FUNCTION_BLOCK EL_Scale (* Scale: output values from its holder -> outputs (break before make); one holder at a time; all off on release or when the module aborts; inputs -> state channel when they change *)
  (* Standard: 61499-2 *)
  (* Version 0.1, 2026-09-28, Project contributors, AAU Smart Production Lab *)
  PACKAGE filling;
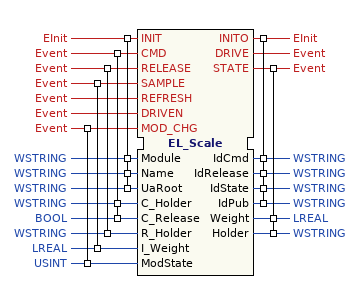
  EVENT_INPUT
    INIT : EInit WITH Module, Name, UaRoot;
    CMD WITH C_Holder, C_Release;
    RELEASE WITH R_Holder;
    SAMPLE WITH I_Weight;
    REFRESH;
    DRIVEN;
    MOD_CHG WITH ModState;
  END_EVENT
  EVENT_OUTPUT
    INITO : EInit WITH IdCmd, IdRelease, IdState, IdPub;
    DRIVE;
    STATE WITH Weight, Holder;
  END_EVENT
  VAR_INPUT
    Module : WSTRING;
    Name : WSTRING;
    UaRoot : WSTRING;
    C_Holder : WSTRING;
    C_Release : BOOL;
    R_Holder : WSTRING;
    I_Weight : LREAL;
    ModState : USINT;
  END_VAR
  VAR_OUTPUT
    IdCmd : WSTRING;
    IdRelease : WSTRING;
    IdState : WSTRING;
    IdPub : WSTRING;
    Weight : LREAL;
    Holder : WSTRING;
  END_VAR
  VAR
    Publish : BOOL;
    Beat : USINT;
    LastHolder : WSTRING;
    Pending : BOOL;
    OffPending : BOOL;
    L_Weight : LREAL;
  END_VAR
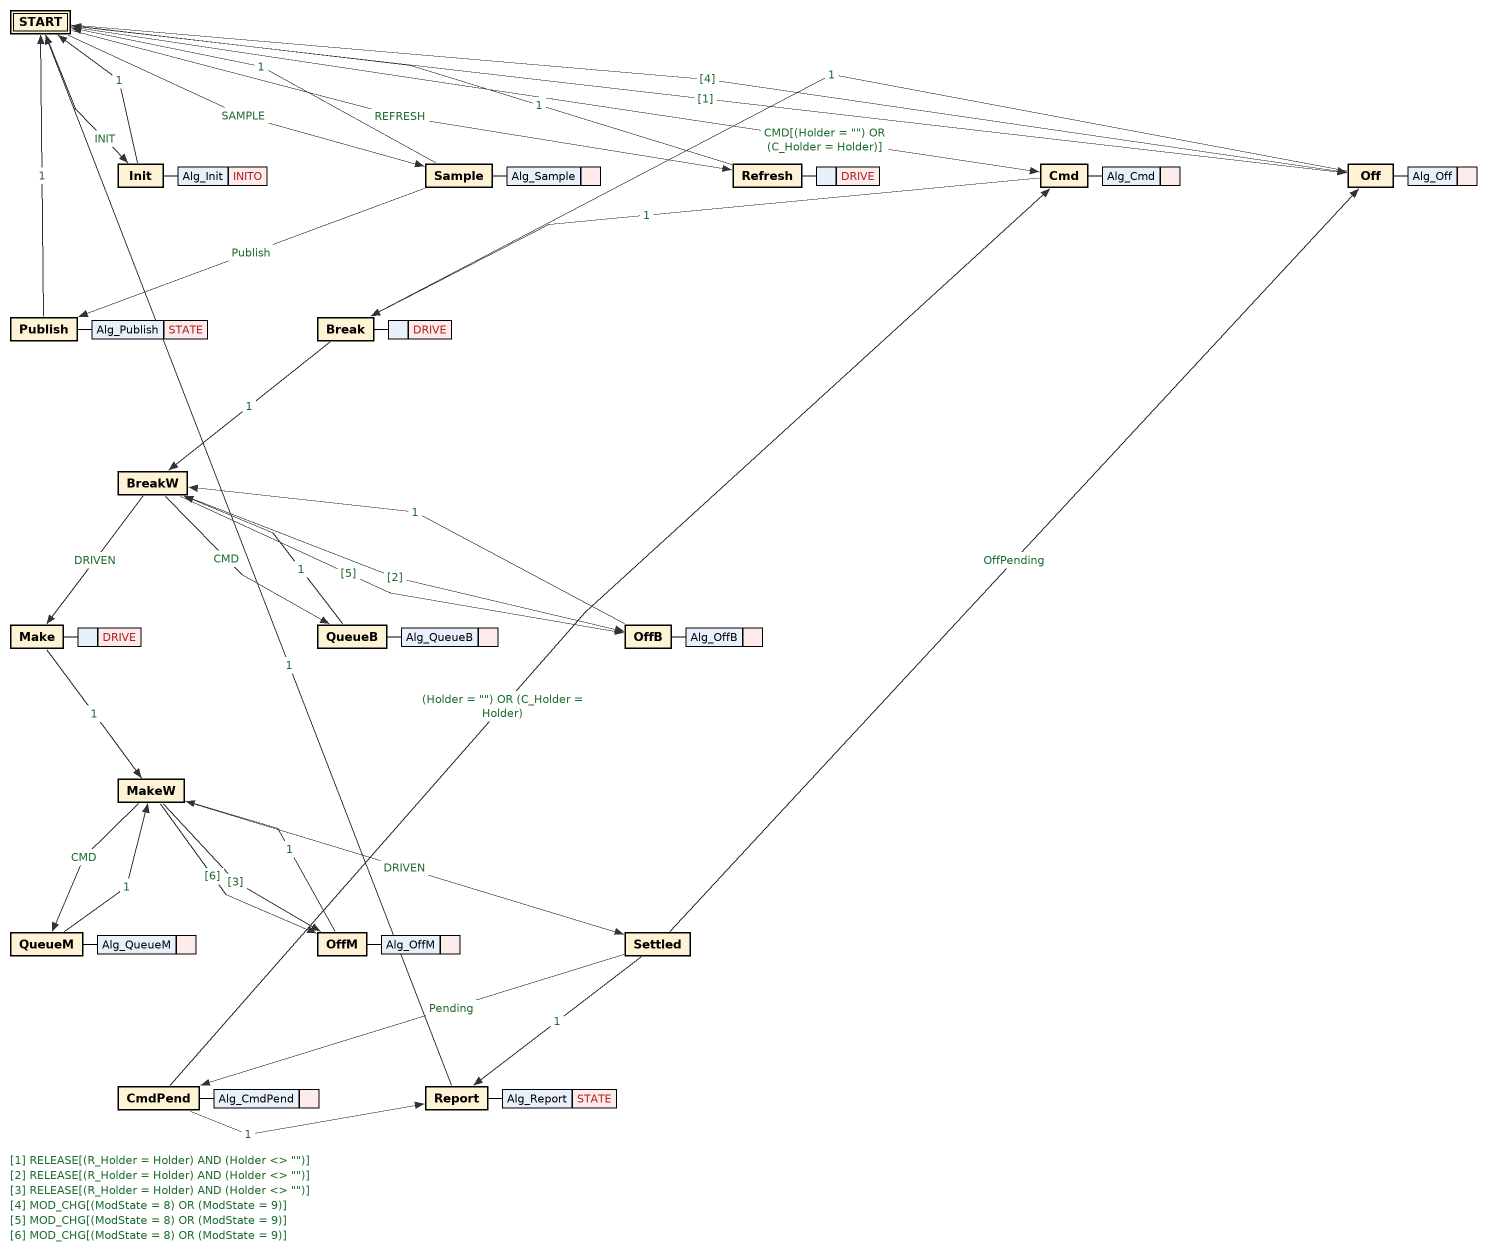
  EC_STATES
    START;
    Init : Alg_Init -> INITO;
    Sample : Alg_Sample;
    Publish : Alg_Publish -> STATE;
    Refresh : -> DRIVE;
    Cmd : Alg_Cmd;
    Off : Alg_Off;
    Break : -> DRIVE;
    Make : -> DRIVE;
    BreakW;
    MakeW;
    QueueB : Alg_QueueB;
    OffB : Alg_OffB;
    QueueM : Alg_QueueM;
    OffM : Alg_OffM;
    CmdPend : Alg_CmdPend;
    Settled;
    Report : Alg_Report -> STATE;
  END_STATES
  EC_TRANSITIONS
    START TO Init := INIT;
    START TO Sample := SAMPLE;
    START TO Refresh := REFRESH;
    START TO Cmd := CMD[(Holder = "") OR (C_Holder = Holder)];
    START TO Off := RELEASE[(R_Holder = Holder) AND (Holder <> "")];
    START TO Off := MOD_CHG[(ModState = 8) OR (ModState = 9)];
    Init TO START := 1;
    Sample TO Publish := Publish;
    Sample TO START := 1;
    Publish TO START := 1;
    Refresh TO START := 1;
    Cmd TO Break := 1;
    Off TO Break := 1;
    Break TO BreakW := 1;
    BreakW TO Make := DRIVEN;
    Make TO MakeW := 1;
    MakeW TO Settled := DRIVEN;
    BreakW TO QueueB := CMD;
    BreakW TO OffB := RELEASE[(R_Holder = Holder) AND (Holder <> "")];
    BreakW TO OffB := MOD_CHG[(ModState = 8) OR (ModState = 9)];
    QueueB TO BreakW := 1;
    OffB TO BreakW := 1;
    MakeW TO QueueM := CMD;
    MakeW TO OffM := RELEASE[(R_Holder = Holder) AND (Holder <> "")];
    MakeW TO OffM := MOD_CHG[(ModState = 8) OR (ModState = 9)];
    QueueM TO MakeW := 1;
    OffM TO MakeW := 1;
    Settled TO Off := OffPending;
    Settled TO CmdPend := Pending;
    CmdPend TO Cmd := (Holder = "") OR (C_Holder = Holder);
    CmdPend TO Report := 1;
    Settled TO Report := 1;
    Report TO START := 1;
  END_TRANSITIONS
  ALGORITHM Alg_Init IN ST:
IdCmd := CONCAT(CONCAT(CONCAT(CONCAT("loc[", Module), "/"), Name), "/cmd]");
IdRelease := CONCAT(CONCAT(CONCAT(CONCAT("loc[", Module), "/"), Name), "/release]");
IdState := CONCAT(CONCAT(CONCAT(CONCAT("loc[", Module), "/"), Name), "/state]");
IdPub := CONCAT(CONCAT(CONCAT(CONCAT(CONCAT("opc_ua[WRITE;", UaRoot), "/Equipment/"), Name), "/Weight"), "]");
  END_ALGORITHM
  ALGORITHM Alg_Sample IN ST:
Weight := I_Weight;
Publish := (Weight <> L_Weight) OR (Holder <> LastHolder) OR (Beat >= 20);
Beat := Beat + 1;
  END_ALGORITHM
  ALGORITHM Alg_Publish IN ST:
L_Weight := Weight;
LastHolder := Holder;
Beat := 0;
  END_ALGORITHM
  ALGORITHM Alg_Cmd IN ST:
Holder := C_Holder;
IF C_Release THEN
  Holder := "";
END_IF;
  END_ALGORITHM
  ALGORITHM Alg_Off IN ST:
Holder := "";
OffPending := FALSE;
  END_ALGORITHM
  ALGORITHM Alg_QueueB IN ST:
Pending := TRUE;
  END_ALGORITHM
  ALGORITHM Alg_OffB IN ST:
OffPending := TRUE;
  END_ALGORITHM
  ALGORITHM Alg_QueueM IN ST:
Pending := TRUE;
  END_ALGORITHM
  ALGORITHM Alg_OffM IN ST:
OffPending := TRUE;
  END_ALGORITHM
  ALGORITHM Alg_CmdPend IN ST:
Pending := FALSE;
  END_ALGORITHM
  ALGORITHM Alg_Report IN ST:
LastHolder := Holder;
Beat := 0;
  END_ALGORITHM
END_FUNCTION_BLOCK
